Fanuc KAREL source: kb00173.KL

-- PROVISIONAL review KL for V770-1; original PC SHA256 86fd98628b967f57ef594e5859b4f292af84475f34fe4a83bbca8a1829dafc2d
-- Incomplete behavior may be omitted. Consult companion uncertainty JSON. Do not deploy.
PROGRAM KB00173
%NOLOCKGROUP
BEGIN
  -- UNRESOLVED_PC offsets 5-12; opcodes 9D,23
  -- UNRESOLVED_PC offsets 17-24; opcodes 9D,23
  -- UNRESOLVED_PC offsets 29-36; opcodes 9D,23
  -- UNRESOLVED_PC offsets 41-48; opcodes 9D,23
  -- UNRESOLVED_PC offsets 53-81; opcodes 27,22,22,22,22,31
  -- UNRESOLVED_PC offsets 86-90; opcodes 7F
END KB00173
